// TIA Portal V20 export
FUNCTION "GenerateTransactionID" : Void   // FC20221, LAD
{ S7_Optimized_Access := 'TRUE' }
// stored: AutoNumber false, SetENOAutomatically false
   VAR_INPUT
      i_Start : Int;
   END_VAR
   VAR_OUTPUT
      dw_TransactionID : DWord;
   END_VAR
   VAR_TEMP
      i_Dummy : Int;
      t_DTL : DTL;
      i_CurrentYear : UInt;
      i_CurrentMonth : USInt;
      i_CurrentDay : USInt;
      i_CurrentHour : USInt;
      i_CurrentMinute : USInt;
      i_CurrentSecond : USInt;
      i_CurrentMilliSecond : UDInt;
      dw_CurrentYearToSecond : DWord;
      dw_CurrentMonthToSecond : DWord;
      dw_CurrentDayToSecond : DWord;
      dw_CurrentHourToSecond : DWord;
      dw_CurrentMinuteToSecond : DWord;
   END_VAR
BEGIN

REGION Network 1: Read time of day
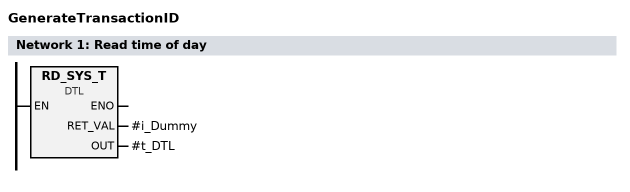
   RUNG wire#powerrail
      { S7_Templates := "date_type := DTL" } RD_SYS_T(RET_VAL => #i_Dummy, OUT => #t_DTL)
   END_RUNG
   // the same network as SCL:
   #i_Dummy := RD_SYS_T(OUT => #t_DTL);
END_REGION

REGION Network 2 (SCL): Generate unique values
   IF #i_Start = 1 THEN
       #i_CurrentYear := #t_DTL.YEAR;
       IF #i_CurrentYear > 1970 THEN
           #i_CurrentYear := #i_CurrentYear - 1970
           ;
       END_IF;//NEW

       #i_CurrentMonth := #t_DTL.MONTH;
       #i_CurrentDay := #t_DTL.DAY;
       #i_CurrentHour := #t_DTL.HOUR;
       #i_CurrentMinute := #t_DTL.MINUTE;
       #i_CurrentSecond := #t_DTL.SECOND;
       #i_CurrentMilliSecond := #t_DTL.NANOSECOND;

       #dw_CurrentYearToSecond := #i_CurrentYear * 31536000;
       #dw_CurrentMonthToSecond := #i_CurrentMonth * 2635200;
       #dw_CurrentDayToSecond := #i_CurrentDay * 86400;
       #dw_CurrentHourToSecond := #i_CurrentHour * 3600;
       #dw_CurrentMinuteToSecond := #i_CurrentMinute * 60;

       #dw_TransactionID := #dw_CurrentYearToSecond;
       #dw_TransactionID := #dw_TransactionID + #dw_CurrentMonthToSecond;
       #dw_TransactionID := #dw_TransactionID + #dw_CurrentDayToSecond;
       #dw_TransactionID := #dw_TransactionID + #dw_CurrentHourToSecond;
       #dw_TransactionID := #dw_TransactionID + #dw_CurrentMinuteToSecond;
       #dw_TransactionID := #dw_TransactionID + #i_CurrentSecond;
       #dw_TransactionID := #dw_TransactionID - #i_CurrentMilliSecond;

       IF #dw_TransactionID > 1620000000 THEN
           #dw_TransactionID := #dw_TransactionID - 1600000000;
       END_IF;

   ELSE
       #dw_TransactionID := 0;

   END_IF;
END_REGION
END_FUNCTION
